INTERFACE I_EnumerableCollection

METHOD PUBLIC DeregisterEnumerator
VAR_INPUT
	Enumerator : I_Enumerator;
END_VAR
END_METHOD

METHOD RegisterEnumerator
VAR_INPUT
	Enumerator : I_Enumerator;
END_VAR
END_METHOD

END_INTERFACE

(* stored: Version 1.1.0.1, ProductVersion 3.1.4024.12
   Itf I_EnumerableCollection: Id {15d3f50c-3579-44cc-8ca9-882d031f1c7f}
   Method DeregisterEnumerator: Id {d1f4fd95-0094-438d-a51a-81effcd4a530}
   Method RegisterEnumerator: Id {af38f441-9079-49f8-87ff-3e711c383c6c} *)
